TYPE E_State :
(
    Init := 0,
    Idle,
	ActivateExtSg,
    Run,
    StoppingSlave,
	StoppingMaster,
    Error,
    Resetting 
);
END_TYPE

(* stored: Version 1.1.0.1
   DUT E_State: Id {09eb885f-2de7-41de-90f6-fd5bd7181c82} *)
